Fanuc KAREL source: kf00102.KL

-- PROVISIONAL review KL for V770-1; original PC SHA256 0dae3d8a30eede46baa232c35906b7b899ac85c230db2ce17317afbf298a70bc
-- Incomplete behavior may be omitted. Consult companion uncertainty JSON. Do not deploy.
PROGRAM KF00102
%NOLOCKGROUP
BEGIN
  -- UNRESOLVED_PC offsets 5-16; opcodes 2E,23
  -- UNRESOLVED_PC offsets 21-32; opcodes 2E,23
  -- UNRESOLVED_PC offsets 37-63; opcodes 27,27,9D,22,1C,22,27,9D,31
  -- UNRESOLVED_PC offsets 68-72; opcodes 7F
END KF00102
